TYPE T_FolderName : STRING[25];
END_TYPE

(* stored: Version 1.1.0.1
   DUT T_FolderName: Id {5ee52976-b056-427a-ba0f-c8508e5b26a1} *)
